{attribute addProperty BoxType "KL2502"}
{attribute addProperty Id "Channel_1Channel_585D17BE00Channel_2Channel_585D17BE00"}
{attribute addProperty CRC "3457887495"}
{attribute addProperty SizeInBites "0"}
{attribute addProperty SizeInBytes "0"}
TYPE KL2502_CE1B2D07 :
STRUCT
	{attribute addProperty Name "Channel_1"}
	Channel_1 : Channel_585D17BE;
	{attribute addProperty Name "Channel_2"}
	Channel_2 : Channel_585D17BE;
END_STRUCT
END_TYPE

(* stored: Version 1.2.0.0, ProductVersion 3.1.4024.9
   DUT KL2502_CE1B2D07: Id {58d8a954-f2bf-4d45-b131-b4dbe6a3e9a9} *)
